KUKA KRL program: ab_st600_r1_1_1.src, ab_st600_r1_1_1.dat

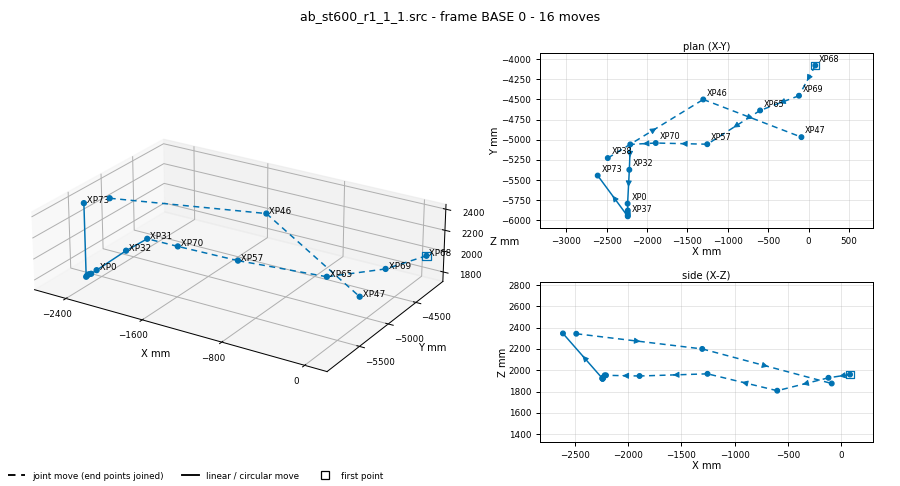
[picture p0: tool path of ab_st600_r1_1_1.src in frame BASE 0, 16 of 17 moves have a stored position in this frame; points joined in program order, loops and branches not executed]
--- ab_st600_r1_1_1.src ---
&ACCESS RVO1
&REL 36
&COMMENT Deposita traseira ACTROS LTA MGS
&PARAM DISKPATH = KRC:\R1\Program
DEF ab_st600_r1_1_1( )
;FOLD INI
  ;FOLD BASISTECH INI
    GLOBAL INTERRUPT DECL 3 WHEN $STOPMESS==TRUE DO IR_STOPM ( )
    INTERRUPT ON 3
    BAS (#INITMOV,0 )
  ;ENDFOLD (BASISTECH INI)
;FOLD GRIPPERTECH INI
USER_GRP(0,DUMMY,DUMMY,GDEFAULT)
;ENDFOLD (GRIPPERTECH INI)
  ;FOLD USER INI
    ;Make your modifications here

  ;ENDFOLD (USER INI)
;ENDFOLD (INI)

; Caracterização dos meios de produção:
; Versão Atual:
; 08/06/2013 12:00 Name: P13.050-R1 CHANGES: Deposita Traseira
; Actros na Geobox LTA\LTB\MGSB\MGS

chk_w5_wechs_ok ( )              ; CHECK GRIPPER ACTROS

;FOLD PTP P68 Vel=100 % PDAT80 Tool[5]:Painel Traseiro Actros Base[0];%{PE}%R 8.2.20,%MKUKATPBASIS,%CMOVE,%VPTP,%P 1:PTP, 2:P68, 3:, 5:100, 7:PDAT80
$BWDSTART=FALSE
PDAT_ACT=PPDAT80
FDAT_ACT=FP68
BAS(#PTP_PARAMS,100)
PTP XP68
;ENDFOLD

;FOLD OUT 3353 'Solicitar lib para entrar com peca geo' State=TRUE ;%{PE}%R 8.2.20,%MKUKATPBASIS,%COUT,%VOUTX,%P 2:3353, 3:Solicitar lib para entrar com peca geo, 5:TRUE, 6:
$OUT[3353]=TRUE
;ENDFOLD
;FOLD WAIT FOR ( IN 3353 'Aguarda lib para entrar com a peca geo' );%{PE}%R 8.2.20,%MKUKATPBASIS,%CEXT_WAIT_FOR,%VEXT_WAIT_FOR,%P 2:, 4:, 5:$IN, 6:3353, 7:Aguarda lib para entrar com a peca geo, 9:
WAIT FOR  ( $IN[3353] )
;ENDFOLD
;FOLD OUT 3353 'Solicitar lib para entrar com peca geo' State=FALSE ;%{PE}%R 8.2.20,%MKUKATPBASIS,%COUT,%VOUTX,%P 2:3353, 3:Solicitar lib para entrar com peca geo, 5:FALSE, 6:
$OUT[3353]=FALSE
;ENDFOLD

;FOLD OUT 3346 'Entrega peça Geo box' State=TRUE ;%{PE}%R 8.2.20,%MKUKATPBASIS,%COUT,%VOUTX,%P 2:3346, 3:Entrega peça Geo box, 5:TRUE, 6:
$OUT[3346]=TRUE
;ENDFOLD
;FOLD WAIT FOR ( IN 3346 'Aguarda lib. Entregar peça Geo box' );%{PE}%R 8.2.20,%MKUKATPBASIS,%CEXT_WAIT_FOR,%VEXT_WAIT_FOR,%P 2:, 4:, 5:$IN, 6:3346, 7:Aguarda lib. Entregar peça Geo box, 9:
WAIT FOR  ( $IN[3346] )
;ENDFOLD
;FOLD OUT 3346 'Entrega peça Geo box' State=FALSE ;%{PE}%R 8.2.20,%MKUKATPBASIS,%COUT,%VOUTX,%P 2:3346, 3:Entrega peça Geo box, 5:FALSE, 6:
$OUT[3346]=FALSE
;ENDFOLD
;FOLD OUT 3348 'Fora area GEOBOX' State=FALSE ;%{PE}%R 8.2.20,%MKUKATPBASIS,%COUT,%VOUTX,%P 2:3348, 3:Fora area GEOBOX, 5:FALSE, 6:
$OUT[3348]=FALSE
;ENDFOLD

;FOLD PTP P69 CONT Vel=100 % PDAT81 Tool[8]:TOOL_CHANGER Base[1]:Actros;%{PE}%R 8.2.20,%MKUKATPBASIS,%CMOVE,%VPTP,%P 1:PTP, 2:P69, 3:C_DIS, 5:100, 7:PDAT81
$BWDSTART=FALSE
PDAT_ACT=PPDAT81
FDAT_ACT=FP69
BAS(#PTP_PARAMS,100)
PTP XP69 C_DIS
;ENDFOLD
;FOLD PTP P65 CONT Vel=100 % PDAT79 Tool[8]:TOOL_CHANGER Base[1]:Actros;%{PE}%R 8.2.20,%MKUKATPBASIS,%CMOVE,%VPTP,%P 1:PTP, 2:P65, 3:C_DIS, 5:100, 7:PDAT79
$BWDSTART=FALSE
PDAT_ACT=PPDAT79
FDAT_ACT=FP65
BAS(#PTP_PARAMS,100)
PTP XP65 C_DIS
;ENDFOLD
;FOLD PTP P57 CONT Vel=100 % PDAT48 Tool[8]:TOOL_CHANGER Base[1]:Actros;%{PE}%R 8.2.20,%MKUKATPBASIS,%CMOVE,%VPTP,%P 1:PTP, 2:P57, 3:C_DIS, 5:100, 7:PDAT48
$BWDSTART=FALSE
PDAT_ACT=PPDAT48
FDAT_ACT=FP57
BAS(#PTP_PARAMS,100)
PTP XP57 C_DIS
;ENDFOLD
;FOLD PTP P70 CONT Vel=100 % PDAT82 Tool[8]:TOOL_CHANGER Base[1]:Actros;%{PE}%R 8.2.20,%MKUKATPBASIS,%CMOVE,%VPTP,%P 1:PTP, 2:P70, 3:C_DIS, 5:100, 7:PDAT82
$BWDSTART=FALSE
PDAT_ACT=PPDAT82
FDAT_ACT=FP70
BAS(#PTP_PARAMS,100)
PTP XP70 C_DIS
;ENDFOLD
;FOLD PTP P31 Vel=100 % PDAT29 Tool[5]:Painel Traseiro Actros Base[0];%{PE}%R 8.2.20,%MKUKATPBASIS,%CMOVE,%VPTP,%P 1:PTP, 2:P31, 3:, 5:100, 7:PDAT29
$BWDSTART=FALSE
PDAT_ACT=PPDAT29
FDAT_ACT=FP31
BAS(#PTP_PARAMS,100)
PTP XP31
;ENDFOLD

;FOLD Collision.Monitoring_AREA_5_Off . ;%{PE}%MKUKATPUSER
COLLSTOP( 11, 2+0 )
;ENDFOLD

;FOLD LIN P32 Vel=0.8 m/s CPDAT6 Tool[5]:Painel Traseiro Actros Base[0];%{PE}%R 8.2.20,%MKUKATPBASIS,%CMOVE,%VLIN,%P 1:LIN, 2:P32, 3:, 5:0.8, 7:CPDAT6
$BWDSTART=FALSE
LDAT_ACT=LCPDAT6
FDAT_ACT=FP32
BAS(#CP_PARAMS,0.8)
LIN XP32
;ENDFOLD
;FOLD LIN P0 Vel=0.8 m/s CPDAT19 Tool[5]:Painel Traseiro Actros Base[0];%{PE}%R 8.2.20,%MKUKATPBASIS,%CMOVE,%VLIN,%P 1:LIN, 2:P0, 3:, 5:0.8, 7:CPDAT19
$BWDSTART=FALSE
LDAT_ACT=LCPDAT19
FDAT_ACT=FP0
BAS(#CP_PARAMS,0.8)
LIN XP0
;ENDFOLD
;FOLD LIN P79 Vel=0.18 m/s CPDAT26 Tool[5]:Painel Traseiro Actros Base[0];%{PE}%R 8.2.20,%MKUKATPBASIS,%CMOVE,%VLIN,%P 1:LIN, 2:P79, 3:, 5:0.18, 7:CPDAT26
$BWDSTART=FALSE
LDAT_ACT=LCPDAT26
FDAT_ACT=FP79
BAS(#CP_PARAMS,0.18)
LIN XP79
;ENDFOLD

;FOLD SET Z3.1/2 GRP ACTROS State=OPN GDAT4;%{PE}%R 8.2.1,%MKUKATPGRP,%CGRP,%VGRP,%P 2:2, 4:1, 5:#NO, 6:GDAT4, 8:0, 10:0
H50(GRP,2,1,GGDAT4)
;ENDFOLD
chk_w5_grp3_opn()

;FOLD LIN P72 Vel=0.4 m/s CPDAT20 Tool[5]:Painel Traseiro Actros Base[0];%{PE}%R 8.2.20,%MKUKATPBASIS,%CMOVE,%VLIN,%P 1:LIN, 2:P72, 3:, 5:0.4, 7:CPDAT20
$BWDSTART=FALSE
LDAT_ACT=LCPDAT20
FDAT_ACT=FP72
BAS(#CP_PARAMS,0.4)
LIN XP72
;ENDFOLD

;FOLD LIN P37 Vel=0.3 m/s CPDAT16 Tool[5]:Painel Traseiro Actros Base[0];%{PE}%R 8.2.20,%MKUKATPBASIS,%CMOVE,%VLIN,%P 1:LIN, 2:P37, 3:, 5:0.3, 7:CPDAT16
$BWDSTART=FALSE
LDAT_ACT=LCPDAT16
FDAT_ACT=FP37
BAS(#CP_PARAMS,0.3)
LIN XP37
;ENDFOLD

;FOLD ; POSICAO DE DEPOSITO DA PECA NA GEOBOX;%{PE}%R 8.2.20,%MKUKATPBASIS,%CCOMMENT,%VNORMAL,%P 2:POSICAO  DE DEPOSITO  DA  PECA  NA  GEOBOX
;ENDFOLD
;FOLD LIN P81 Vel=0.3 m/s CPDAT28 Tool[5]:Painel Traseiro Actros Base[0];%{PE}%R 8.2.20,%MKUKATPBASIS,%CMOVE,%VLIN,%P 1:LIN, 2:P81, 3:, 5:0.3, 7:CPDAT28
$BWDSTART=FALSE
LDAT_ACT=LCPDAT28
FDAT_ACT=FP81
BAS(#CP_PARAMS,0.3)
LIN XP81
;ENDFOLD

;FOLD OUT 3345 'Solicita lib sair da geo box' State=TRUE ;%{PE}%R 8.2.20,%MKUKATPBASIS,%COUT,%VOUTX,%P 2:3345, 3:Solicita lib sair da geo box, 5:TRUE, 6:
$OUT[3345]=TRUE
;ENDFOLD
;FOLD WAIT FOR ( IN 3344 'Aguarda lib. sair geo box' );%{PE}%R 8.2.20,%MKUKATPBASIS,%CEXT_WAIT_FOR,%VEXT_WAIT_FOR,%P 2:, 4:, 5:$IN, 6:3344, 7:Aguarda lib. sair geo box, 9:
WAIT FOR  ( $IN[3344] )
;ENDFOLD
;FOLD OUT 3345 'Solicita lib sair da geo box' State=FALSE ;%{PE}%R 8.2.20,%MKUKATPBASIS,%COUT,%VOUTX,%P 2:3345, 3:Solicita lib sair da geo box, 5:FALSE, 6:
$OUT[3345]=FALSE
;ENDFOLD
;FOLD OUT 3344 'R1 Entregou peca geo box' State=FALSE ;%{PE}%R 8.2.20,%MKUKATPBASIS,%COUT,%VOUTX,%P 2:3344, 3:R1 Entregou peca geo box, 5:FALSE, 6:
$OUT[3344]=FALSE
;ENDFOLD

;FOLD OUT 2 'Vacuo - Válvula de vácuo para ventosas S1.1 / S1.2 / S1.3 / S1.4 - Actros Todos'  State= FALSE;%{PE}%R 8.2.17,%MKUKATPBASIS,%COUT,%VOUTX,%P 2:2, 3:Vacuo - Válvula de vácuo para ventosas S1.1 / S1.2 / S1.3 / S1.4 - Actros Todos, 5:FALSE, 6:

$OUT[2]=FALSE
;ENDFOLD
;FOLD PULSE 3 'Expulsar - Válvula de vácuo para ventosas S1.1 / S1.2 / S1.3 / S1.4 - Actros Todos' State=TRUE Time=1 sec;%{PE}%R 8.2.20,%MKUKATPBASIS,%COUT,%VPULSE,%P 2:3, 3:Expulsar - Válvula de vácuo para ventosas S1.1 / S1.2 / S1.3 / S1.4 - Actros Todos, 5:TRUE, 6:, 8:1
PULSE($OUT[3], TRUE,1)
;ENDFOLD

;FOLD SET Z3.1/2 GRP ACTROS State=CLO GDAT2;%{PE}%R 8.2.1,%MKUKATPGRP,%CGRP,%VGRP,%P 2:2, 4:2, 5:#NO, 6:GDAT2, 8:0, 10:0
H50(GRP,2,2,GGDAT2)
;ENDFOLD
chk_w5_grp3_clo()

;FOLD OUT 224 'Bloquear MPS' State=FALSE ;%{PE}%R 8.2.20,%MKUKATPBASIS,%COUT,%VOUTX,%P 2:224, 3:Bloquear MPS, 5:FALSE, 6:
$OUT[224]=FALSE
;ENDFOLD
;FOLD OUT 223 'Desbloquear MPS' State=TRUE ;%{PE}%R 8.2.20,%MKUKATPBASIS,%COUT,%VOUTX,%P 2:223, 3:Desbloquear MPS, 5:TRUE, 6:
$OUT[223]=TRUE
;ENDFOLD
;FOLD WAIT FOR ( IN 217 'MPS Destravado' );%{PE}%R 8.2.20,%MKUKATPBASIS,%CEXT_WAIT_FOR,%VEXT_WAIT_FOR,%P 2:, 4:, 5:$IN, 6:217, 7:MPS Destravado, 9:
WAIT FOR  ( $IN[217] )
;ENDFOLD
;FOLD WAIT FOR NOT ( IN 221 'MPS Travado' );%{PE}%R 8.2.20,%MKUKATPBASIS,%CEXT_WAIT_FOR,%VEXT_WAIT_FOR,%P 2:NOT, 4:, 5:$IN, 6:221, 7:MPS Travado, 9:
WAIT FOR  NOT ( $IN[221] )
;ENDFOLD
;FOLD WAIT Time=0.5 sec;%{PE}%R 8.2.20,%MKUKATPBASIS,%CWAIT,%VWAIT,%P 3:0.5
WAIT SEC 0.5
;ENDFOLD
;FOLD IBUS OFF;%{PE}%R 8.2.20,%MKUKATPBASIS,%CIBUS,%VMAP,%P 2:#OFF, 3:1
$IBUS_OFF=$IBUS_ON
$IBUS_ON=0
;ENDFOLD
;FOLD WAIT Time=0.25 sec;%{PE}%R 8.2.20,%MKUKATPBASIS,%CWAIT,%VWAIT,%P 3:0.25
WAIT SEC 0.25
;ENDFOLD

;FOLD LIN P73 Vel=0.3 m/s CPDAT21 Tool[8]:TOOL_CHANGER Base[0];%{PE}%R 8.2.20,%MKUKATPBASIS,%CMOVE,%VLIN,%P 1:LIN, 2:P73, 3:, 5:0.3, 7:CPDAT21
$BWDSTART=FALSE
LDAT_ACT=LCPDAT21
FDAT_ACT=FP73
BAS(#CP_PARAMS,0.3)
LIN XP73
;ENDFOLD
;FOLD LIN P77 CONT Vel=0.5 m/s CPDAT24 Tool[8]:TOOL_CHANGER Base[1]:Actros;%{PE}%R 8.2.20,%MKUKATPBASIS,%CMOVE,%VLIN,%P 1:LIN, 2:P77, 3:C_DIS C_DIS, 5:0.5, 7:CPDAT24
$BWDSTART=FALSE
LDAT_ACT=LCPDAT24
FDAT_ACT=FP77
BAS(#CP_PARAMS,0.5)
LIN XP77 C_DIS C_DIS
;ENDFOLD

;FOLD PTP P38 Vel=100 % PDAT85 Tool[8]:TOOL_CHANGER Base[0];%{PE}%R 8.2.20,%MKUKATPBASIS,%CMOVE,%VPTP,%P 1:PTP, 2:P38, 3:, 5:100, 7:PDAT85
$BWDSTART=FALSE
PDAT_ACT=PPDAT85
FDAT_ACT=FP38
BAS(#PTP_PARAMS,100)
PTP XP38
;ENDFOLD

;FOLD WAIT FOR NOT ( IN 219 'Posicao p/ Acoplamento OK' );%{PE}%R 8.2.20,%MKUKATPBASIS,%CEXT_WAIT_FOR,%VEXT_WAIT_FOR,%P 2:NOT, 4:, 5:$IN, 6:219, 7:Posicao p/ Acoplamento OK, 9:
WAIT FOR  NOT ( $IN[219] )
;ENDFOLD
;FOLD OUT 223 'Desbloquear MPS' State=FALSE ;%{PE}%R 8.2.20,%MKUKATPBASIS,%COUT,%VOUTX,%P 2:223, 3:Desbloquear MPS, 5:FALSE, 6:
$OUT[223]=FALSE
;ENDFOLD
;FOLD OUT 3349 'R1 Pegou peca' State=FALSE ;%{PE}%R 8.2.20,%MKUKATPBASIS,%COUT,%VOUTX,%P 2:3349, 3:R1 Pegou peca, 5:FALSE, 6:
$OUT[3349]=FALSE
;ENDFOLD
;FOLD OUT 3344 'R1 entregou peça geo box' State=FALSE ;%{PE}%R 8.2.20,%MKUKATPBASIS,%COUT,%VOUTX,%P 2:3344, 3:R1 entregou peça geo box, 5:FALSE, 6:
$OUT[3344]=FALSE
;ENDFOLD
;FOLD OUT 3348 'Fora area GEOBOX' State=TRUE ;%{PE}%R 8.2.20,%MKUKATPBASIS,%COUT,%VOUTX,%P 2:3348, 3:Fora area GEOBOX, 5:TRUE, 6:
$OUT[3348]=TRUE
;ENDFOLD
;FOLD OUT 3344 'R1 entregou peça geo box' State=TRUE ;%{PE}%R 8.2.20,%MKUKATPBASIS,%COUT,%VOUTX,%P 2:3344, 3:R1 entregou peça geo box, 5:TRUE, 6:
$OUT[3344]=TRUE
;ENDFOLD

;FOLD PTP P46 CONT Vel=100 % PDAT37 Tool[8]:TOOL_CHANGER Base[1]:Actros;%{PE}%R 8.2.20,%MKUKATPBASIS,%CMOVE,%VPTP,%P 1:PTP, 2:P46, 3:C_DIS, 5:100, 7:PDAT37
$BWDSTART=FALSE
PDAT_ACT=PPDAT37
FDAT_ACT=FP46
BAS(#PTP_PARAMS,100)
PTP XP46 C_DIS
;ENDFOLD
;FOLD PTP P47 CONT Vel=100 % PDAT38 Tool[8]:TOOL_CHANGER Base[1]:Actros;%{PE}%R 8.2.20,%MKUKATPBASIS,%CMOVE,%VPTP,%P 1:PTP, 2:P47, 3:C_DIS, 5:100, 7:PDAT38
$BWDSTART=FALSE
PDAT_ACT=PPDAT38
FDAT_ACT=FP47
BAS(#PTP_PARAMS,100)
PTP XP47 C_DIS
;ENDFOLD

;FOLD OUT 3344 'R1 entregou peça geo box' State=FALSE ;%{PE}%R 8.2.20,%MKUKATPBASIS,%COUT,%VOUTX,%P 2:3344, 3:R1 entregou peça geo box, 5:FALSE, 6:
$OUT[3344]=FALSE
;ENDFOLD
END

--- ab_st600_r1_1_1.dat ---
&ACCESS RVO1
&REL 36
&COMMENT Deposita traseira ACTROS LTA MGS
&PARAM DISKPATH = KRC:\R1\Program
DEFDAT  ab_st600_r1_1_1
;FOLD EXTERNAL DECLARATIONS;%{PE}%MKUKATPBASIS,%CEXT,%VCOMMON,%P
;FOLD GRIPPERTECH EXT
EXT  H50 (INT  :IN,INT  :IN,INT  :IN,GRP_TYP  :IN )
;ENDFOLD (GRIPPERTECH EXT)
;FOLD SPOTTECH EXT

;ENDFOLD (SPOTTECH EXT)
;FOLD BASISTECH EXT;%{PE}%MKUKATPBASIS,%CEXT,%VEXT,%P
EXT  BAS (BAS_COMMAND  :IN,REAL  :IN )
DECL INT SUCCESS
;ENDFOLD (BASISTECH EXT)
;FOLD USER EXT;%{E}%MKUKATPUSER,%CEXT,%VEXT,%P
;Make your modifications here

;ENDFOLD (USER EXT)
;ENDFOLD (EXTERNAL DECLARATIONS)

;# ============ START PATH : bh_p13050r1_lta_01 =============
DECL BASIS_SUGG_T LAST_BASIS={POINT1[] "P0                      ",POINT2[] "P0                      ",CP_PARAMS[] "CPDAT0                  ",PTP_PARAMS[] "PDAT0                   ",CONT[] "                        ",CP_VEL[] "0.3                     ",PTP_VEL[] "100                     ",SYNC_PARAMS[] "SYNCDAT                 ",SPL_NAME[] "S0                      "}
DECL E6POS XP31={X -2208.68994,Y -5057.91113,Z 1952.19104,A -88.9759293,B 89.2573166,C 2.63928199,S 2,T 10,E1 -4321.06787,E2 0.0,E3 0.0,E4 0.0,E5 0.0,E6 0.0}
DECL FDAT FP31={TOOL_NO 5,BASE_NO 0,IPO_FRAME #BASE,POINT2[] " ",TQ_STATE FALSE}
DECL PDAT PPDAT29={VEL 100.0,ACC 100.0,APO_DIST 100.0,APO_MODE #CDIS}
DECL E6POS XP32={X -2220.66309,Y -5372.58496,Z 1952.18701,A -88.9353027,B 89.2573471,C 2.67988205,S 2,T 10,E1 -4321.06787,E2 0.0,E3 0.0,E4 0.0,E5 0.0,E6 0.0}
DECL FDAT FP32={TOOL_NO 5,BASE_NO 0,IPO_FRAME #BASE,POINT2[] " ",TQ_STATE FALSE}
DECL LDAT LCPDAT6={VEL 2.0,ACC 100.0,APO_DIST 100.0,APO_FAC 50.0,AXIS_VEL 100.0,AXIS_ACC 100.0,ORI_TYP #VAR,CIRC_TYP #BASE,JERK_FAC 50.0,GEAR_JERK 50.0,EXAX_IGN 0}
DECL E6POS XP37={X -2239.7439,Y -5936.67822,Z 1926.62695,A -100.503197,B 88.9303436,C -10.5974503,S 2,T 10,E1 -4320.28613,E2 0.0,E3 0.0,E4 0.0,E5 0.0,E6 0.0}
DECL FDAT FP37={TOOL_NO 5,BASE_NO 0,IPO_FRAME #BASE,POINT2[] " ",TQ_STATE FALSE}
DECL E6POS XP38={X -2487.7251,Y -5227.0498,Z 2342.58789,A -27.4018593,B -75.25914,C 87.3958664,S 2,T 10,E1 -4320.27393,E2 0.0,E3 0.0,E4 0.0,E5 0.0,E6 0.0}
DECL FDAT FP38={TOOL_NO 8,BASE_NO 0,IPO_FRAME #BASE,POINT2[] " ",TQ_STATE FALSE}
DECL E6POS XP46={X -1304.44397,Y -4500.89307,Z 2199.95898,A 62.3853683,B 34.4934082,C -142.184601,S 2,T 10,E1 -4318.39307,E2 0.0,E3 0.0,E4 0.0,E5 0.0,E6 0.0}
DECL FDAT FP46={TOOL_NO 8,BASE_NO 0,IPO_FRAME #BASE,POINT2[] " ",TQ_STATE FALSE}
DECL PDAT PPDAT37={VEL 100.0,ACC 100.0,APO_DIST 100.0,APO_MODE #CDIS}
DECL E6POS XP47={X -88.1010895,Y -4967.96289,Z 1875.21399,A -59.9045906,B -3.67260695,C 176.441299,S 2,T 2,E1 -3477.44312,E2 0.0,E3 0.0,E4 0.0,E5 0.0,E6 0.0}
DECL FDAT FP47={TOOL_NO 8,BASE_NO 0,IPO_FRAME #BASE,POINT2[] " ",TQ_STATE FALSE}
DECL PDAT PPDAT38={VEL 100.0,ACC 100.0,APO_DIST 100.0,APO_MODE #CDIS}
DECL E6POS XP57={X -1254.78296,Y -5055.70313,Z 1965.95996,A -4.48244905,B 88.810112,C 90.8473892,S 2,T 10,E1 -4246.70801,E2 0.0,E3 0.0,E4 0.0,E5 0.0,E6 0.0}
DECL FDAT FP57={TOOL_NO 5,BASE_NO 0,IPO_FRAME #BASE,POINT2[] " ",TQ_STATE FALSE}
DECL PDAT PPDAT48={VEL 100.0,ACC 100.0,APO_DIST 10.0,APO_MODE #CDIS}
DECL GRP_SUGG_T LAST_GRP={NUMBER[] "2                       ",STATE[] "1                       ",PARAMS[] "GDAT2                   "}
DECL GRP_TYP GGDAT1={G_APO #NO,GRP_TIME 0.200000003,CTRL #OFF,DLY 0,DST 1}
DECL GRP_TYP GCONT={G_APO #YES,GRP_TIME 0.0,CTRL #OFF,DLY 0,DST 0}
DECL GRP_TYP GGDAT3={G_APO #NO,GRP_TIME 0.200000003,CTRL #OFF,DLY 0,DST 1}
DECL GRP_TYP GGDAT2={G_APO #NO,GRP_TIME 0.200000003,CTRL #OFF,DLY 0,DST 1}
DECL LDAT LCPDAT16={VEL 2.0,ACC 100.0,APO_DIST 100.0,APO_FAC 50.0,AXIS_VEL 100.0,AXIS_ACC 100.0,ORI_TYP #VAR,CIRC_TYP #BASE,JERK_FAC 50.0,GEAR_JERK 50.0,EXAX_IGN 0}
DECL E6POS XP65={X -599.781677,Y -4637.07324,Z 1807.53198,A 89.7495117,B 80.6197968,C 177.934402,S 2,T 10,E1 -3056.61792,E2 0.0,E3 0.0,E4 0.0,E5 0.0,E6 0.0}
DECL FDAT FP65={TOOL_NO 5,BASE_NO 0,IPO_FRAME #BASE,POINT2[] " ",TQ_STATE FALSE}
DECL PDAT PPDAT79={VEL 100.0,ACC 100.0,APO_DIST 100.0,APO_MODE #CDIS}
DECL LDAT LCPDAT19={VEL 2.0,ACC 100.0,APO_DIST 100.0,APO_FAC 50.0,AXIS_VEL 100.0,AXIS_ACC 100.0,ORI_TYP #VAR,CIRC_TYP #BASE,JERK_FAC 50.0,GEAR_JERK 50.0,EXAX_IGN 0}
DECL E6POS XP0={X -2242.04199,Y -5791.70703,Z 1920.72705,A -103.606598,B 89.4271317,C -13.5311804,S 2,T 10,E1 -4320.27393,E2 0.0,E3 0.0,E4 0.0,E5 0.0,E6 0.0}
DECL FDAT FP0={TOOL_NO 5,BASE_NO 0,IPO_FRAME #BASE,POINT2[] " ",TQ_STATE FALSE}
DECL E6POS XP68={X 83.9785233,Y -4080.4231,Z 1959.36597,A 36.8050804,B 88.5113831,C 81.7786865,S 2,T 10,E1 -2701.98999,E2 0.0,E3 0.0,E4 0.0,E5 0.0,E6 0.0}
DECL FDAT FP68={TOOL_NO 5,BASE_NO 0,IPO_FRAME #BASE,POINT2[] " ",TQ_STATE FALSE}
DECL PDAT PPDAT80={VEL 100.0,ACC 100.0,APO_DIST 100.0,APO_MODE #CDIS}
DECL E6POS XP69={X -118.355499,Y -4454.77881,Z 1928.73499,A 84.1095428,B 89.4634018,C 147.737,S 2,T 10,E1 -2873.82397,E2 0.0,E3 0.0,E4 0.0,E5 0.0,E6 0.0}
DECL FDAT FP69={TOOL_NO 5,BASE_NO 0,IPO_FRAME #BASE,POINT2[] " ",TQ_STATE FALSE}
DECL PDAT PPDAT81={VEL 100.0,ACC 100.0,APO_DIST 100.0,APO_MODE #CDIS}
DECL E6POS XP70={X -1893.21899,Y -5040.83984,Z 1945.64697,A 102.737198,B 88.6551971,C -164.3237,S 2,T 10,E1 -4289.93506,E2 0.0,E3 0.0,E4 0.0,E5 0.0,E6 0.0}
DECL FDAT FP70={TOOL_NO 5,BASE_NO 0,IPO_FRAME #BASE,POINT2[] " ",TQ_STATE FALSE}
DECL PDAT PPDAT82={VEL 100.0,ACC 100.0,APO_DIST 10.0,APO_MODE #CDIS}
DECL E6POS XP72={X -2239.81909,Y -5910.29395,Z 1928.46106,A -84.2885971,B 89.2003784,C 5.914186,S 2,T 10,E1 -4320.28711,E2 0.0,E3 0.0,E4 0.0,E5 0.0,E6 0.0}
DECL FDAT FP72={TOOL_NO 5,BASE_NO 0,IPO_FRAME #BASE,POINT2[] " ",TQ_STATE FALSE}
DECL LDAT LCPDAT20={VEL 2.0,ACC 100.0,APO_DIST 100.0,APO_FAC 50.0,AXIS_VEL 100.0,AXIS_ACC 100.0,ORI_TYP #VAR,CIRC_TYP #BASE,JERK_FAC 50.0,GEAR_JERK 50.0,EXAX_IGN 0}
DECL E6POS XP73={X -2612.7019,Y -5444.20313,Z 2345.48511,A -27.4024696,B -75.2591629,C 87.3966827,S 2,T 10,E1 -4320.27393,E2 0.0,E3 0.0,E4 0.0,E5 0.0,E6 0.0}
DECL FDAT FP73={TOOL_NO 8,BASE_NO 0,IPO_FRAME #BASE,POINT2[] " ",TQ_STATE FALSE}
DECL LDAT LCPDAT21={VEL 2.0,ACC 50.0,APO_DIST 100.0,APO_FAC 50.0,AXIS_VEL 100.0,AXIS_ACC 100.0,ORI_TYP #VAR,CIRC_TYP #BASE,JERK_FAC 50.0,GEAR_JERK 50.0,EXAX_IGN 0}
DECL PDAT PPDAT85={VEL 100.0,ACC 100.0,APO_DIST 100.0,APO_MODE #CDIS}
DECL E6POS XP77={X 2866.18994,Y -232.274902,Z 837.087891,A -117.401901,B -75.25914,C 87.3958664,S 2,T 10,E1 -4320.27393,E2 0.0,E3 0.0,E4 0.0,E5 0.0,E6 0.0}
DECL FDAT FP77={TOOL_NO 8,BASE_NO 1,IPO_FRAME #BASE,POINT2[] " ",TQ_STATE FALSE}
DECL LDAT LCPDAT24={VEL 2.0,ACC 100.0,APO_DIST 100.0,APO_FAC 50.0,AXIS_VEL 100.0,AXIS_ACC 100.0,ORI_TYP #VAR,CIRC_TYP #BASE,JERK_FAC 50.0,GEAR_JERK 50.0,EXAX_IGN 0}
DECL E6POS XP79={X -2239.78101,Y -5876.91699,Z 1920.14795,A -90.9768066,B 89.2029419,C -1.06975102,S 2,T 10,E1 -4320.28516,E2 0.0,E3 0.0,E4 0.0,E5 0.0,E6 0.0}
DECL FDAT FP79={TOOL_NO 5,BASE_NO 0,IPO_FRAME #BASE,POINT2[] " ",TQ_STATE FALSE}
DECL LDAT LCPDAT26={VEL 2.0,ACC 100.0,APO_DIST 100.0,APO_FAC 50.0,AXIS_VEL 100.0,AXIS_ACC 100.0,ORI_TYP #VAR,CIRC_TYP #BASE,JERK_FAC 50.0,GEAR_JERK 50.0,EXAX_IGN 0}
DECL E6POS XP81={X -2240.07104,Y -5949.60205,Z 1920.15601,A -99.7001572,B 89.2208328,C -9.53020477,S 2,T 10,E1 -4320.28906,E2 0.0,E3 0.0,E4 0.0,E5 0.0,E6 0.0}
DECL FDAT FP81={TOOL_NO 5,BASE_NO 0,IPO_FRAME #BASE,POINT2[] " ",TQ_STATE FALSE}
DECL LDAT LCPDAT28={VEL 2.0,ACC 100.0,APO_DIST 100.0,APO_FAC 50.0,AXIS_VEL 100.0,AXIS_ACC 100.0,ORI_TYP #VAR,CIRC_TYP #BASE,JERK_FAC 50.0,GEAR_JERK 50.0,EXAX_IGN 0}
DECL GRP_TYP GGDAT4={G_APO #NO,GRP_TIME 0.200000003,CTRL #OFF,DLY 0,DST 1}
DECL GRP_TYP GGDAT5={G_APO #NO,GRP_TIME 0.200000003,CTRL #OFF,DLY 0,DST 1}
ENDDAT
